// TIA Portal V17 export
// export: Created 2025-06-26T07:49:46.3250842Z, ExportSetting WithDefaults, DisplayName Totally Integrated Automation Portal, DisplayVersion V17 Update 8, DisplayName TIA Portal Openness, DisplayVersion V17 Update 8, DisplayName TIA Portal Version Control Interface, DisplayVersion V17, DisplayName STEP 7 Professional, DisplayVersion V17 Update 8, DisplayName STEP 7 Safety, DisplayVersion V17 Update 6, DisplayName WinCC Advanced, DisplayVersion V17 Update 8
FUNCTION "fcPID_Regulator" : Void   // FC54, FBD
{ S7_Optimized_Access := 'TRUE' }
VERSION : 0.1
// stored: AutoNumber true, IsIECCheckEnabled false, SetENOAutomatically false, UDAEnableTagReadback false
   VAR_INPUT
      ControllerDeviation : Real;
      Kp : Real;
      Tn : Real;
      Tv : Real;
      "T1_MAX_0,25s" : Real;
      LowerLimit : Real;
      UpperLimit : Real;
      ManualTrigger : Bool;
      ManualValue : Real;
      fCycleTime : Real;
   END_VAR
   VAR_OUTPUT
      Output : Real;
      LowerLimit_Reached : Bool;
      UpperLimit_Reached : Bool;
   END_VAR
   VAR_IN_OUT
      LastDT1_Memory : Real;
      IntegralPart_Memory : Real;
      ParameterChange_Memory : Real;
   END_VAR
   VAR_TEMP
      DifferentialFactor : Real;
      DT1 : Real;
      ProportionalPart : Real;
      "PI-Part" : Real;
      ResetFactor : Real;
   END_VAR
BEGIN

REGION Network 1 (SCL): Controller difference and calculation of proportional part
   #ProportionalPart := (#ControllerDeviation) * #Kp;
END_REGION

REGION Network 2 (SCL): DT1 formular
   #DT1 :=(#ControllerDeviation - #LastDT1_Memory) / (#"T1_MAX_0,25s" + #fCycleTime);

   //Stores Merk for the DT1 calculation of the next cycle
   #LastDT1_Memory += #DT1 * #fCycleTime;
END_REGION

REGION Network 3 (SCL): Calculation of the differential part factor
   // Reset Differential part if Tv=0 or ManaulValue active or DifferentialFactor=NAN or if Kp was changed
   IF #Tv = 0 OR #ManualTrigger OR "isNaN"(#DT1) THEN
       #DifferentialFactor := 0;
       #LastDT1_Memory := 0;
   ELSE
       #DifferentialFactor := #DT1 * #Kp * #Tv;
   END_IF;
END_REGION

REGION Network 4 (SCL): Calculation of the integral part
   // Reset Integal memory if Tn=0 or if IntegralPart_Memory=NaN
   IF (#Tn <> 0) AND "isNotNaN"(#IntegralPart_Memory) THEN
   //The integral part is calculated by the last integral part
       #IntegralPart_Memory +=           
       //plus the propotional part devided by the integral factor
       #ProportionalPart * (#fCycleTime / #Tn) -
       //in case of parameter changes on Kp an improving value must be substracted to balance the changes on Kp
       #ControllerDeviation * (#Kp - #ParameterChange_Memory);
   ELSE
       //Deactivates the integral part, if there's no valid number at Tn
       #IntegralPart_Memory := 0;
   END_IF;
END_REGION

REGION Network 5 (SCL): Combination of integral, proportional and differential parts and limit monitoring and switch to manual value
   #"PI-Part" := #ProportionalPart + #IntegralPart_Memory;

   IF #ManualTrigger THEN
       #Output := #ManualValue;
   ELSE
       //Limiting OutputValue to given limits
       #Output := LIMIT(MN := #LowerLimit, IN := #"PI-Part" + #DifferentialFactor, MX := #UpperLimit);
       //Show if a limit got reached
       #LowerLimit_Reached := NOT (#Output > #LowerLimit);
       #UpperLimit_Reached := #Output >= #UpperLimit;
   END_IF;
END_REGION

REGION Network 6 (SCL): Choice of feedback variable (wind up prevention) and calculation of the integral part
   #ResetFactor := (#fCycleTime / (#Tn+0.001)) * 3;// Factor between 1 and oo. 1 compensates Integral and stops sum to grow above maximum. Faktor 500 Sum is limited to match upper boundary after 1/20 Tn

   IF #ManualTrigger THEN
       //feeds back a manual-value-depending value, which is close to be constant and protects the controller against wind up
       #IntegralPart_Memory := #ManualValue - #ProportionalPart;
   ELSIF #"PI-Part" > #UpperLimit THEN
       //feeds back a upper-limit-depending value, which is close to be constant and protects the controller against wind up
       //#IntegralPart_Memory := #UpperLimit - #ProportionalPart;
       #IntegralPart_Memory += (#UpperLimit - #ProportionalPart) * #ResetFactor;
       #IntegralPart_Memory /= 1 + #ResetFactor;
   ELSIF #"PI-Part" < #LowerLimit THEN
       //feeds back a lower-limit-depending value, which is close to be constant and protects the controller against wind up
       //#IntegralPart_Memory := #LowerLimit - #ProportionalPart;
       #IntegralPart_Memory += (#LowerLimit - #ProportionalPart) * #ResetFactor;
       #IntegralPart_Memory /= 1 + #ResetFactor;
   END_IF;

   //If the Kp parameter is changing the integral part gets adjusted to it. Therefore the last Kp value must be stored for the next cycle
   #ParameterChange_Memory := #Kp;
END_REGION
END_FUNCTION
